(* CODESYS project proldPou.export

Project tree, tasks and I/O mapping:
  program POU [ST]
*)

// POU
PROGRAM POU

VAR
    tonGenTimer  : TON; // The "Heartbeat" timer
    tpSensorHold : TP;  // Holds the sensor on 


END_VAR


IF GVL.xSystemRunning THEN

    // 1.  Heartbeat: Fires every 4 seconds
    tonGenTimer(IN := NOT tonGenTimer.Q, PT := T#4S);
    
    // 2. The "Stretcher": Catches the heartbeat and stays ON for 1 solid second
    tpSensorHold(IN := tonGenTimer.Q, PT := T#1S);
    
    // 3. Cycle the Item Type (1 -> 2 -> 3)
    IF tonGenTimer.Q THEN
        GVL.iItemType := GVL.iItemType + 1;
        IF GVL.iItemType > 3 THEN 
            GVL.iItemType := 1; 
        END_IF
    END_IF
    
    // 4. Turn the correct sensor ON
    IF tpSensorHold.Q THEN
        CASE GVL.iItemType OF
            1: 
                GVL.xSensor1 := TRUE;
                GVL.xSensor2 := FALSE;
                GVL.xSensor3 := FALSE;
            2: 
                GVL.xSensor1 := FALSE;
                GVL.xSensor2 := TRUE;
                GVL.xSensor3 := FALSE;
            3: 
                GVL.xSensor1 := FALSE;
                GVL.xSensor2 := FALSE;
                GVL.xSensor3 := TRUE;
        END_CASE
    ELSE
        GVL.xSensor1 := FALSE;
        GVL.xSensor2 := FALSE;
        GVL.xSensor3 := FALSE;
    END_IF

ELSE
    // IF THE SYSTEM IS OFF: Reset everything
    tonGenTimer(IN := FALSE, PT := T#4S);
    tpSensorHold(IN := FALSE, PT := T#1S);
    GVL.xSensor1 := FALSE;
    GVL.xSensor2 := FALSE;
    GVL.xSensor3 := FALSE;
END_IF

END_PROGRAM
